TYPE ST_PowerHeaterSys :
STRUCT
END_STRUCT
END_TYPE

(* stored: Version 1.1.0.1, ProductVersion 3.1.4024.12
   DUT ST_PowerHeaterSys: Id {1d8df876-4613-4377-8be6-608115da678b} *)
